FUNCTION_BLOCK ToWin32ErrorCode_Tests EXTENDS TcUnit.FB_TestSuite

ConversionOfValidErrorCode();

METHOD ConversionOfValidErrorCode
TcUnit.TEST('ConversionOfValidErrorCode');

AssertEquals_UDINT(
    Expected:=Win32ErrorCodes.ERROR_FILE_EXISTS,
    Actual:=ToWin32ErrorCode(80),
    Message:='Error conversion not correct.'
);

TcUnit.TEST_FINISHED();
END_METHOD

END_FUNCTION_BLOCK

(* stored: Version 1.1.0.1, ProductVersion 3.1.4024.11
   POU ToWin32ErrorCode_Tests: Id {642d2499-70f1-4caf-86fe-53406ef48db3}, SpecialFunc None
   Method ConversionOfValidErrorCode: Id {e4b8f277-05e1-427d-8433-5540129e6254} *)
